// TIA Portal V16 export
// export: Created 2022-11-17T15:49:09.4724221Z, ExportSetting WithDefaults, DisplayName Totally Integrated Automation Portal, DisplayVersion V16 Update 6, DisplayName TIA Portal Version Control Interface, DisplayVersion V16 Update 2, DisplayName TIA Portal Openness, DisplayVersion V16 Update 6, DisplayName SINAMICS Startdrive Advanced, DisplayVersion V16 Update 5, DisplayName SINAMICS Startdrive G130, G150, S120, S150, SINAMICS MV, S210, DisplayVersion V16 Update 5, DisplayName SINAMICS Startdrive G110M, G120, G120C, G120D, G120P, G115D, DisplayVersion V16 Update 5, DisplayName STEP 7 Professional, DisplayVersion V16 Update 6, DisplayName STEP 7 Safety, DisplayVersion V16, DisplayName WinCC Advanced, DisplayVersion V16 Update 6
FUNCTION_BLOCK "Modbus"   // FB20, FBD
{ S7_Optimized_Access := 'FALSE' }
VERSION : 0.1
// stored: AutoNumber false, IsIECCheckEnabled false, SetENOAutomatically false, UDAEnableTagReadback false
   VAR_INPUT
      BAUDRATE : UDInt := 115200;
      HW_ID : PORT := 272;
      RESP_TO : UInt := 1000;
      CYCLIC_PROCESSING : Bool := true;
      MB_ADDR : UInt := 8;
      DATA_AD_R : UDInt := 40001;
      DATA_AD_W : UDInt := 40006;
      DATA_LEN_R : UInt := 5;
      DATA_LEN_W : UInt := 5;
      ReadOnly : Bool := 1;   // Read only (1)
   END_VAR
   VAR_OUTPUT
      ERROR : Bool;
      ERROR_INFO : Struct
         drive_number : USInt;
         "step" : USInt;
         STATUS : Word;
      END_STRUCT;
   END_VAR
   VAR_IN_OUT
      ReadDone_0 : Bool;   // Read done for prestretch board (1)
      DT_PTR_IN : Variant;
      DT_PTR_OUT : Variant;
   END_VAR
   VAR DB_SPECIFIC
      drive_index : USInt := 1;
      "step" : USInt := 0;
      REQ : Bool;
      extended_restart : Bool;
      start_internal : Bool;
   END_VAR
   VAR
      MB_COMM_LOAD_Instance { S7_SetPoint := 'True'} : MB_COMM_LOAD;
      MB_MASTER_Instance { S7_SetPoint := 'True'} : MB_MASTER;
   END_VAR
   VAR_TEMP
      _DONE : Bool;
      _ERROR : Bool;
      _STATUS : Word;
      _cyclic_processing : Bool;
   END_VAR
   VAR_TEMP   // added for the SCL form of the ladder/FBD networks
      _w1 : Bool;
      _w2 : Bool;
      _w3 : Bool;
   END_VAR
BEGIN

REGION Network 1: First cycle
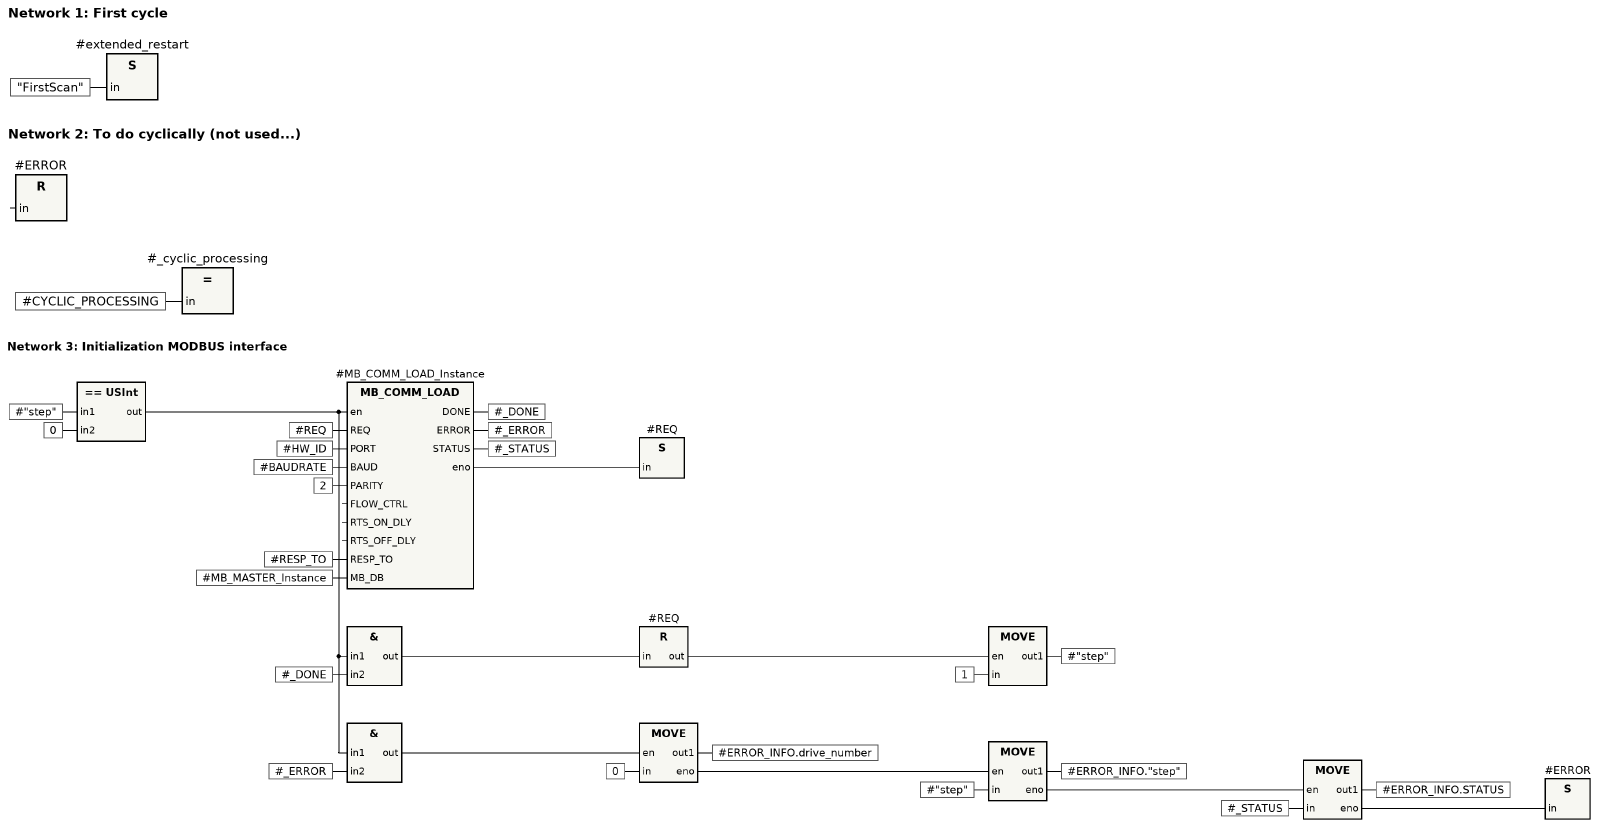
   IF "FirstScan" THEN #extended_restart := TRUE; END_IF;
END_REGION

REGION Network 2: To do cyclically (not used...)
   #ERROR := FALSE;
   #_cyclic_processing := #CYCLIC_PROCESSING;
END_REGION

REGION Network 3: Initialization MODBUS interface
   // ENO of a box is taken as its EN; it also drops when the box reports an error
   #_w1 := #"step" = 0;
   #MB_COMM_LOAD_Instance(EN := #_w1,   // MB_COMM_LOAD
                          REQ := #REQ,
                          PORT := #HW_ID,
                          BAUD := #BAUDRATE,
                          PARITY := 2,
                          RESP_TO := #RESP_TO,
                          MB_DB := #MB_MASTER_Instance,
                          DONE => #_DONE,
                          ERROR => #_ERROR,
                          STATUS => #_STATUS,
                          ENO => #_w2);
   IF #_w2 THEN #REQ := TRUE; END_IF;
   IF #_w1 AND #_DONE THEN
       #REQ := FALSE;
       #"step" := 1;
   END_IF;
   IF #_w1 AND #_ERROR THEN
       #ERROR_INFO.drive_number := 0;
       #ERROR_INFO."step" := #"step";
       #ERROR_INFO.STATUS := #_STATUS;
       #ERROR := TRUE;
   END_IF;
END_REGION

REGION Network 4: READ
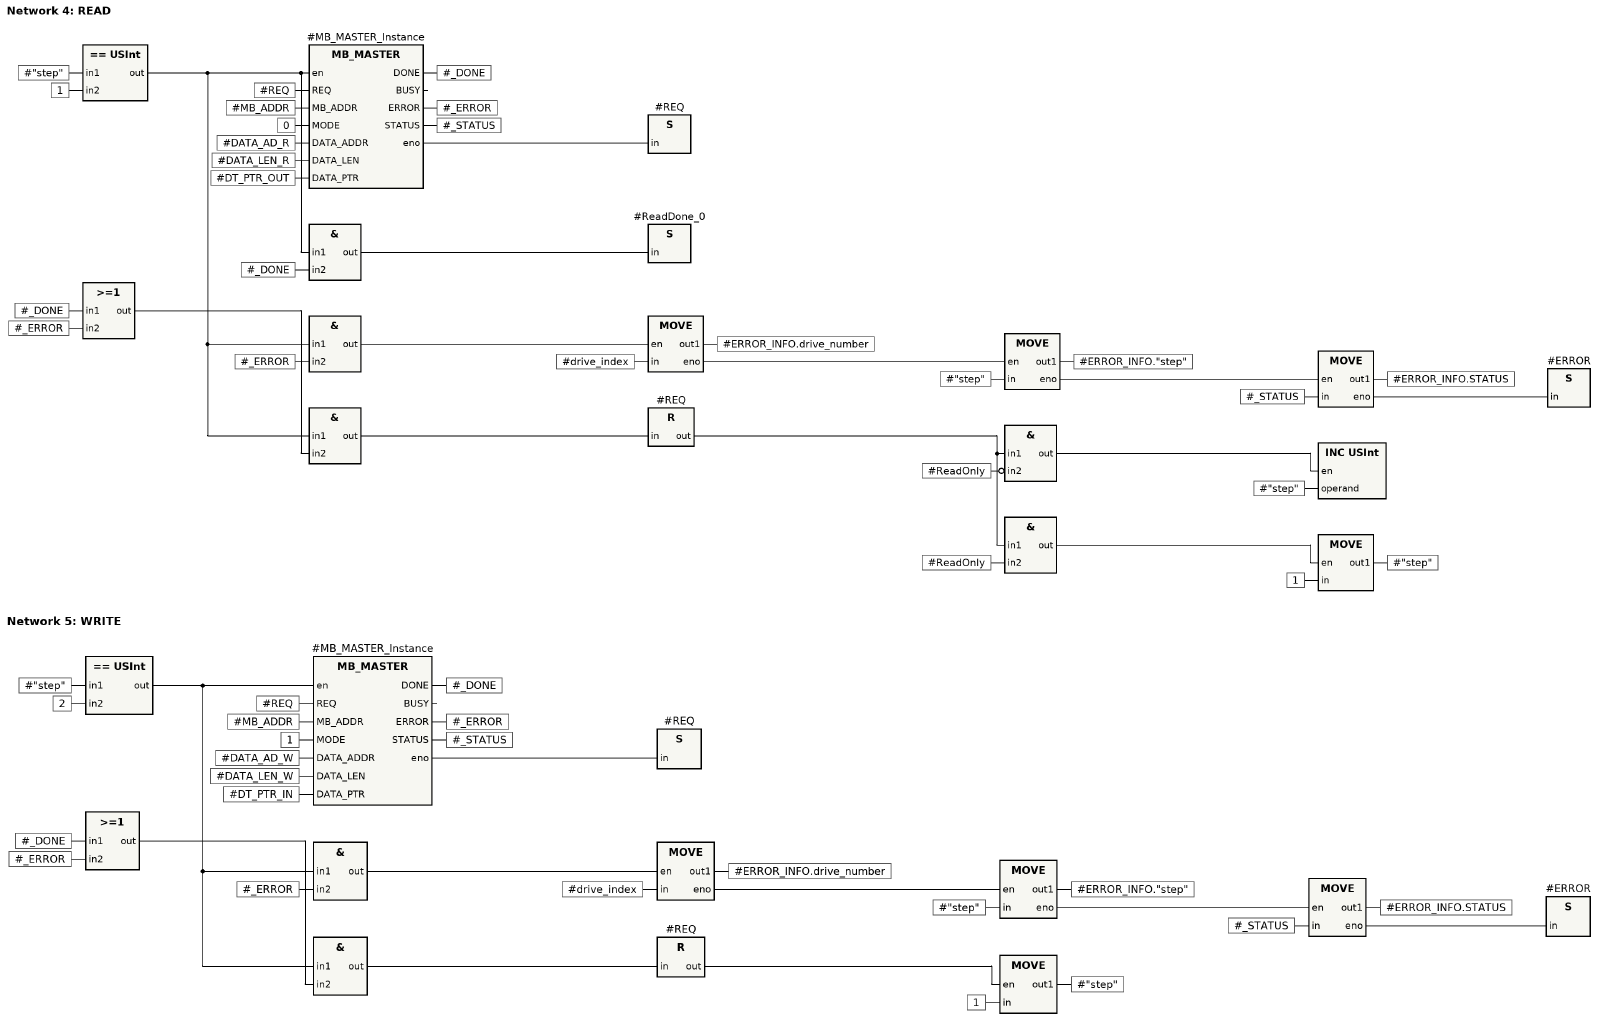
   // ENO of a box is taken as its EN; it also drops when the box reports an error
   #_w1 := #"step" = 1;
   #MB_MASTER_Instance(EN := #_w1,   // MB_MASTER
                       REQ := #REQ,
                       MB_ADDR := #MB_ADDR,
                       MODE := 0,
                       DATA_ADDR := #DATA_AD_R,
                       DATA_LEN := #DATA_LEN_R,
                       DATA_PTR := #DT_PTR_OUT,
                       DONE => #_DONE,
                       ERROR => #_ERROR,
                       STATUS => #_STATUS,
                       ENO => #_w2);
   IF #_w2 THEN #REQ := TRUE; END_IF;
   IF #_w1 AND #_DONE THEN #ReadDone_0 := TRUE; END_IF;
   IF #_w1 AND #_ERROR THEN
       #ERROR_INFO.drive_number := #drive_index;
       #ERROR_INFO."step" := #"step";
       #ERROR_INFO.STATUS := #_STATUS;
       #ERROR := TRUE;
   END_IF;
   #_w3 := #_w1 AND (#_DONE OR #_ERROR);
   IF #_w3 THEN #REQ := FALSE; END_IF;
   IF #_w3 AND NOT #ReadOnly THEN #"step" := #"step" + 1; END_IF;
   IF #_w3 AND #ReadOnly THEN #"step" := 1; END_IF;
END_REGION

REGION Network 5: WRITE
   // ENO of a box is taken as its EN; it also drops when the box reports an error
   #_w1 := #"step" = 2;
   #MB_MASTER_Instance(EN := #_w1,   // MB_MASTER
                       REQ := #REQ,
                       MB_ADDR := #MB_ADDR,
                       MODE := 1,
                       DATA_ADDR := #DATA_AD_W,
                       DATA_LEN := #DATA_LEN_W,
                       DATA_PTR := #DT_PTR_IN,
                       DONE => #_DONE,
                       ERROR => #_ERROR,
                       STATUS => #_STATUS,
                       ENO => #_w2);
   IF #_w2 THEN #REQ := TRUE; END_IF;
   IF #_w1 AND #_ERROR THEN
       #ERROR_INFO.drive_number := #drive_index;
       #ERROR_INFO."step" := #"step";
       #ERROR_INFO.STATUS := #_STATUS;
       #ERROR := TRUE;
   END_IF;
   IF #_w1 AND (#_DONE OR #_ERROR) THEN
       #REQ := FALSE;
       #"step" := 1;
   END_IF;
END_REGION
END_FUNCTION_BLOCK
